PROGRAM MAIN
VAR
END_VAR

MR3K4_KBO_VFS_1(
	i_xPMPS_OK:= TRUE, 
	i_xExt_OK:= TRUE, 
	i_sDevName:= 'TV1K4:VFS:1',
	io_fbFFHWO:= g_FastFaultOutput3
);

(*FastFaultOuput*)	
g_FastFaultOutput3.Execute(bAutoReset:= TRUE);

END_PROGRAM

(* stored: Version 1.1.0.1, ProductVersion 3.1.4024.2
   POU MAIN: Id {4f7257db-fdb3-49ae-b8f5-2bdfa11c0c42}, SpecialFunc None *)
